// TIA Portal project "PLCII_Pro5" (V15.1)

(* hardware
DEVICE "S7-1200 station_1"  S7-1200 Station
   slot 0: "Rack_0"  S7-1200 Rack  Rack  V1.0
   slot 1: "PLC_1"  CPU 1215C DC/DC/Rly  6ES7 215-1HG40-0XB0  V4.2
*)

// ===== PLC "PLC_1"  CPU 1215C DC/DC/Rly =====

VAR_GLOBAL   // PLC tag table "Default tag table"
   "Start" AT %M0.0 : Bool;
   "Sys_runing" AT %M0.1 : Bool;
   "Stop" AT %M0.2 : Bool;
   "Activate" AT %M0.3 : Bool;
   "Sys_Activated" AT %M0.4 : Bool;
END_VAR

DATA_BLOCK "TImerLogic_DB"   // DB1
{ S7_Optimized_Access := 'TRUE' }
VERSION : 0.1
// stored: InstanceOfName TImerLogic
"TImerLogic"
BEGIN
END_DATA_BLOCK

DATA_BLOCK "Rotameter"   // DB2
{ S7_Optimized_Access := 'TRUE' }
VERSION : 0.1
   VAR
      RotameterSig : Bool;
      Flow : Real;
      CounterINT : Real;
      FlowRateGPM : Real;
   END_VAR
BEGIN
END_DATA_BLOCK

FUNCTION_BLOCK "TImerLogic"   // FB1, LAD
{ S7_Optimized_Access := 'TRUE' }
VERSION : 0.1
   VAR
      IEC_Timer_0_Instance : TON_TIME;
      ons1 : Bool;
      ons2 : Bool;
      TimerPT : Time;
      ons3 : Bool;
   END_VAR
   VAR_TEMP   // added for the SCL form of the ladder/FBD networks
      _w1 : Bool;
      _w2 : Bool;
   END_VAR
BEGIN

REGION Network 1
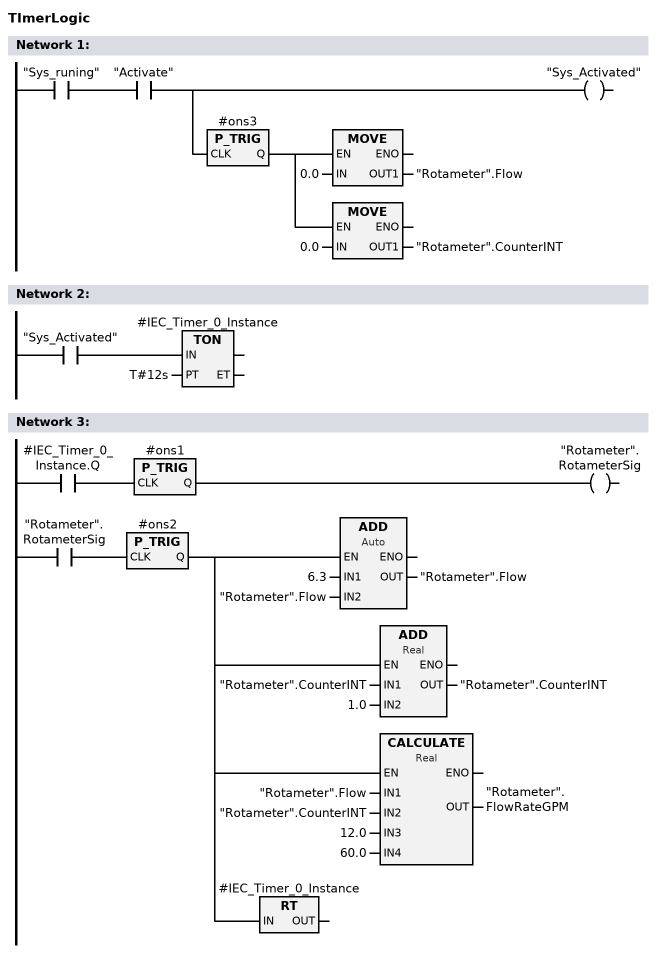
   RUNG wire#powerrail
      Contact( "Sys_runing" )
      Contact( "Activate" )
      wire#w1
      Coil( "Sys_Activated" )
   END_RUNG
   RUNG wire#w1
      P_Trig( #ons3 )
      wire#w2
      Move(in := 0.0, out1 => "Rotameter".Flow)
   END_RUNG
   RUNG wire#w2
      Move(in := 0.0, out1 => "Rotameter".CounterINT)
   END_RUNG
   // the same network as SCL:
   "Sys_Activated" := "Sys_runing" AND "Activate";
   #_w1 := "Sys_Activated" AND NOT #ons3;   // rising edge
   #ons3 := "Sys_Activated";
   IF #_w1 THEN
       "Rotameter".Flow := 0.0;
       "Rotameter".CounterINT := 0.0;
   END_IF;
END_REGION

REGION Network 2
   #IEC_Timer_0_Instance(IN := "Sys_Activated", PT := T#12s);   // TON
END_REGION

REGION Network 3
   RUNG wire#powerrail
      Contact( #IEC_Timer_0_Instance.Q )
      P_Trig( #ons1 )
      Coil( "Rotameter".RotameterSig )
   END_RUNG
   RUNG wire#powerrail
      Contact( "Rotameter".RotameterSig )
      P_Trig( #ons2 )
      wire#w1
      Add(in1 := 6.3, in2 := "Rotameter".Flow, out => "Rotameter".Flow)
   END_RUNG
   RUNG wire#w1
      { S7_Templates := "SrcType := Real" } Add(in1 := "Rotameter".CounterINT, in2 := 1.0, out => "Rotameter".CounterINT)
   END_RUNG
   RUNG wire#w1
      { S7_Templates := "SrcType := Real"; S7_Expression := "((IN1)/(IN3*IN2))*IN4" } Calculate(in1 := "Rotameter".Flow, in2 := "Rotameter".CounterINT, in3 := 12.0, in4 := 60.0, out => "Rotameter".FlowRateGPM)
   END_RUNG
   RUNG wire#w1
      RT_Coil( #IEC_Timer_0_Instance )
   END_RUNG
   // the same network as SCL:
   #_w1 := #IEC_Timer_0_Instance.Q AND NOT #ons1;   // rising edge
   #ons1 := #IEC_Timer_0_Instance.Q;
   "Rotameter".RotameterSig := #_w1;
   #_w2 := "Rotameter".RotameterSig AND NOT #ons2;   // rising edge
   #ons2 := "Rotameter".RotameterSig;
   IF #_w2 THEN
       "Rotameter".Flow := 6.3 + "Rotameter".Flow;
       "Rotameter".CounterINT := "Rotameter".CounterINT + 1.0;
       "Rotameter".FlowRateGPM := (("Rotameter".Flow)/(12.0*"Rotameter".CounterINT))*60.0;
       RESET_TIMER(#IEC_Timer_0_Instance);
   END_IF;
END_REGION
END_FUNCTION_BLOCK

ORGANIZATION_BLOCK "Main"   // OB1, LAD, ProgramCycle
TITLE = "Main Program Sweep (Cycle)"
{ S7_Optimized_Access := 'TRUE' }
VERSION : 0.1
   VAR_INPUT
      Initial_Call : Bool;   // Initial call of this OB
      Remanence : Bool;   // =True, if remanent data are available
   END_VAR
BEGIN

REGION Network 1
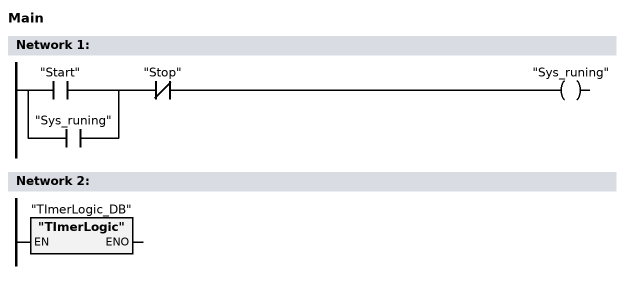
   RUNG wire#powerrail
      Contact( "Start" )
      wire#w1
      I_Contact( "Stop" )
      Coil( "Sys_runing" )
   END_RUNG
   RUNG wire#powerrail
      Contact( "Sys_runing" )
   END_RUNG wire#w1
   // the same network as SCL:
   "Sys_runing" := ("Start" OR "Sys_runing") AND NOT "Stop";
END_REGION

REGION Network 2
   RUNG wire#powerrail
      "TImerLogic_DB"()
   END_RUNG
   // the same network as SCL:
   "TImerLogic_DB"();   // "TImerLogic"
END_REGION
END_ORGANIZATION_BLOCK